TEXTLIST txlTestTypes
  0 = 'none'
  10 = 'EOL'
  20 = 'Performance'
  30 = 'Hour'
  40 = 'Whole'
  50 = 'Cyclic 30'
  60 = 'Cyclic 70'
   = ''
END_TEXTLIST

(* stored: Version 1.1.0.1, ProductVersion 3.1.4024.12
   TextList txlTestTypes: Id {3d2208d1-0ff7-4e5a-b18b-093027a7d30b} *)
